{attribute 'GeneratedUsingTerminal: EK1100-0000-0018'}
{attribute addProperty BoxType "EK1100-0000-0018"}
{attribute addProperty Id "Beckhoff_ELM37xxEK1122Beckhoff_ELM37xxEK1122_0A3745332A_0001_ELM3702_0000_0016ELM3702_73CCAB7A50A_0002_ELM3702_0000_0017ELM3702_73CCAB7A50A_0003_ELM3704_0000_0016ELM3704_7474644C72A_0004_ELM3704_0000_0017ELM3704_7474644C72A_0005_ELM3704_0001_0017ELM3704_7474644C72A_0006_ELM3704_0020_0016ELM3704_7474644C72A_0007_ELM3702_0101_0016ELM3702_73CCAB7A50A_0008_ELM3704_1001_0016ELM3704_7474644C72A_0009_ELM3704_1001_0017ELM3704_7474644C72"}
{attribute addProperty CRC "287287766"}
{attribute addProperty Size "584"}
TYPE Beckhoff_ELM37xx_111FA9D6 EXTENDS EK1100_AB5A9467 :
STRUCT
	{attribute addProperty Name "Beckhoff_ELM37xxEK1122"}
	{attribute addProperty PreviousPort "Beckhoff ELM37xx : B"}
	Beckhoff_ELM37xxEK1122 : Beckhoff_ELM37xxEK1122_0A374533;
	{attribute addProperty Name "A_0001_ELM3702_0000_0016"}
	{attribute addProperty PreviousPort "Beckhoff ELM37xxEK1122 : C"}
	A_0001_ELM3702_0000_0016 : ELM3702_73CCAB7A;
	{attribute addProperty Name "A_0002_ELM3702_0000_0017"}
	{attribute addProperty PreviousPort "A_0001(ELM3702-0000-0016) : B"}
	A_0002_ELM3702_0000_0017 : ELM3702_73CCAB7A;
	{attribute addProperty Name "A_0003_ELM3704_0000_0016"}
	{attribute addProperty PreviousPort "A_0002(ELM3702-0000-0017) : B"}
	A_0003_ELM3704_0000_0016 : ELM3704_7474644C;
	{attribute addProperty Name "A_0004_ELM3704_0000_0017"}
	{attribute addProperty PreviousPort "A_0003(ELM3704-0000-0016) : B"}
	A_0004_ELM3704_0000_0017 : ELM3704_7474644C;
	{attribute addProperty Name "A_0005_ELM3704_0001_0017"}
	{attribute addProperty PreviousPort "A_0004(ELM3704-0000-0017) : B"}
	A_0005_ELM3704_0001_0017 : ELM3704_7474644C;
	{attribute addProperty Name "A_0006_ELM3704_0020_0016"}
	{attribute addProperty PreviousPort "A_0005(ELM3704-0001-0017) : B"}
	A_0006_ELM3704_0020_0016 : ELM3704_7474644C;
	{attribute addProperty Name "A_0007_ELM3702_0101_0016"}
	{attribute addProperty PreviousPort "A_0006(ELM3704-0020-0016) : B"}
	A_0007_ELM3702_0101_0016 : ELM3702_73CCAB7A;
	{attribute addProperty Name "A_0008_ELM3704_1001_0016"}
	{attribute addProperty PreviousPort "A_0007(ELM3702-0101-0016) : B"}
	A_0008_ELM3704_1001_0016 : ELM3704_7474644C;
	{attribute addProperty Name "A_0009_ELM3704_1001_0017"}
	{attribute addProperty PreviousPort "A_0008(ELM3704-1001-0016) : B"}
	A_0009_ELM3704_1001_0017 : ELM3704_7474644C;
END_STRUCT
END_TYPE

(* stored: Version 1.2.0.0, ProductVersion 3.1.4024.9
   DUT Beckhoff_ELM37xx_111FA9D6: Id {98cdc14a-2e5b-475d-9070-7ca1b7a59424} *)
